FUNCTION_BLOCK GENERATEFLIMAGE (* generate flot image *)
  (* Version 1.0, AN, SWDC RTSoft *)
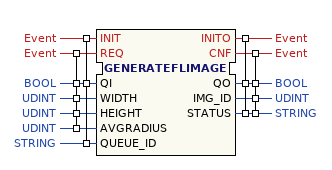
  EVENT_INPUT
    INIT WITH QI, QUEUE_ID;
    REQ WITH QI, WIDTH, HEIGHT, AVGRADIUS;
  END_EVENT
  EVENT_OUTPUT
    INITO WITH QO, STATUS;
    CNF WITH QO, IMG_ID, STATUS;
  END_EVENT
  VAR_INPUT
    QI : BOOL;
    WIDTH : UDINT;
    HEIGHT : UDINT;
    AVGRADIUS : UDINT;
    QUEUE_ID : STRING;
  END_VAR
  VAR_OUTPUT
    QO : BOOL;
    IMG_ID : UDINT;
    STATUS : STRING;
  END_VAR
END_FUNCTION_BLOCK
